// TIA Portal V17 export
// export: Created 2024-08-29T18:23:49.7382109Z, ExportSetting WithDefaults, DisplayName Totally Integrated Automation Portal, DisplayVersion V17 Update 7, DisplayName TIA Portal Openness, DisplayVersion V17 Update 7, DisplayName TIA Portal Version Control Interface, DisplayVersion V17, DisplayName SINAMICS Startdrive Advanced, DisplayVersion V17 SP2, DisplayName SINAMICS Startdrive G110M, G120, G120C, G120D, G120P, G115D, DisplayVersion V17 SP2, DisplayName SINAMICS Startdrive G130, G150, S120, S150, SINAMICS MV, S210, DisplayVersion V17 SP2, DisplayName STEP 7 Professional, DisplayVersion V17 Update 7, DisplayName STEP 7 Safety, DisplayVersion V17 Update 6, DisplayName WinCC Advanced / Unified PC, DisplayVersion V17 Update 7
VAR_GLOBAL   // PLC tag table "Default tag table"
   OutputPin2 AT %QB147 : Byte;
   Tag_2 AT %QB152 : Byte;
   Tag_3 AT %QB155 : Byte;
   Tag_4 AT %QB154 : Byte;
   Tag_5 AT %QB153 : Byte;
   System_Byte AT %MB0 : Byte;
   DiagStatusUpdate AT %M0.1 : Bool;
   Tag_6 AT %MW122 : UInt;
END_VAR
